// Gets the length of a string;
FUNCTION F_StrLen : T_Size
VAR_INPUT
	pString : POINTER TO STRING;
END_VAR
VAR
	i : T_Size := 0;
END_VAR

IF pString = 0 THEN RETURN; END_IF
WHILE pString^[i] <> 0 DO
	i := i + 1;
	END_WHILE
F_StrLen := i;

END_FUNCTION

(* stored: Version 1.1.0.1, ProductVersion 3.1.4024.4
   POU F_StrLen: Id {874be76a-bfe9-4c44-98f5-eacf801fe0ff}, SpecialFunc None *)
